PROGRAM Robot
VAR
	fbRobot						: FB_Robot_Mitsubishi;
	nCurrentState				: DINT;
	nLastState					: DINT;				
	rtRobot_ProgramStarted		: TON;
	rtRobot_ProgramCompleted	: TON;
	fbTimerRobot				:TON;
	gbTimerTimeoutRobot			:TON;
END_VAR

	Stations.gstRobotMitsubishi.sRobotAddress := '192.168.0.20';
	//gstRobotMitsubishi.bAutomaticMode := NOT IO_CONVEYOR.iMAINTENANCE_KEY;
	fbRobot(Robot := Stations.gstRobotMitsubishi,
		PacketManager := Stations.gstRobotMitsubishiPacketManager);
		
rtRobot_ProgramStarted(IN:=NOT Stations.gstRobotMitsubishi.bReady 
						AND NOT Stations.gstRobotMitsubishi.bProgramCompleted, PT:=T#50MS);
rtRobot_ProgramCompleted(IN:= Stations.gstRobotMitsubishi.bReady AND Stations.gstRobotMitsubishi.bProgramCompleted 
							AND Stations.gstRobotMitsubishi.nDependencyState = 0, PT:=T#10MS);

// If robot error
IF Stations.gstRobotMitsubishi.bError AND nCurrentState > E_RobotStates.STATE_INIT_CHECK_ROBOT_ERROR_DONE 
AND nCurrentState < E_RobotStates.STATE_ERROR THEN
	nLastState:=nCurrentState;
	nCurrentState:=E_RobotStates.STATE_ERROR;
END_IF
		
CASE nCurrentState OF
	E_RobotStates.STATE_WAITING_FOR_INIT:
		IF Stations.roboData = dataRequestRobot.roboInit THEN			
			nLastState := nCurrentState;
			nCurrentState := E_RobotStates.STATE_INIT_ROBOT_TOGGLE;
		END_IF
		
	E_RobotStates.STATE_INIT_ROBOT_TOGGLE:
		IF Stations.gstRobotMitsubishi.bAutomaticMode THEN
			Stations.gstRobotMitsubishi.bDoReset:=FALSE;
			Stations.gstRobotMitsubishi.bToggleConnect:=FALSE;
			Stations.gstRobotMitsubishi.bDoStart:=FALSE;
			fbTimerRobot(IN:=TRUE,PT:=T#1000MS);
			IF fbTimerRobot.Q THEN
				fbTimerRobot(IN:=FALSE);				
				nLastState := nCurrentState;
				nCurrentState :=E_RobotStates.STATE_INIT_ROBOT_ON;
			END_IF
		ELSE
			// Robot Auto  = true
		END_IF

	E_RobotStates.STATE_INIT_ROBOT_ON:
		IF Stations.gstRobotMitsubishi.bOnline THEN
			nLastState := nCurrentState;
			nCurrentState :=E_RobotStates.STATE_INIT_CHECK_ROBOT_ERROR;
		ELSE
			Stations.gstRobotMitsubishi.bToggleConnect:=TRUE;
			a_ToggleRobot();
		END_IF	

	E_RobotStates.STATE_INIT_CHECK_ROBOT_ERROR:
		IF Stations.gstRobotMitsubishi.bError OR Stations.gstRobotMitsubishi.nCurrentState = E_Robot_Mitsubishi_States.STATE_WAITING_RESET THEN
			Stations.gstRobotMitsubishi.bDoReset:=TRUE;
			nLastState := nCurrentState;
			nCurrentState :=E_RobotStates.STATE_INIT_CHECK_ROBOT_ERROR_DONE;
		ELSE
			nLastState := nCurrentState;
			nCurrentState :=E_RobotStates.STATE_INIT_CHECK_ROBOT_READY;
		END_IF	
	
	E_RobotStates.STATE_INIT_CHECK_ROBOT_ERROR_DONE:
		IF Stations.gstRobotMitsubishi.nCurrentState = E_Robot_Mitsubishi_States.STATE_OPERATIONAL THEN
			IF NOT Stations.gstRobotMitsubishi.bError THEN
				nLastState := nCurrentState;
				nCurrentState :=E_RobotStates.STATE_INIT_CHECK_ROBOT_READY;
			ELSE
				a_ToggleRobot();
			END_IF
		ELSIF Stations.gstRobotMitsubishi.nCurrentState = E_Robot_Mitsubishi_States.STATE_WAITING_RESET THEN
			nLastState := nCurrentState;
			nCurrentState :=E_RobotStates.STATE_INIT_CHECK_ROBOT_ERROR;
		END_IF
		
	E_RobotStates.STATE_INIT_CHECK_ROBOT_READY:
		IF NOT Stations.gstRobotMitsubishi.bReady OR NOT Stations.gstRobotMitsubishi.bExecuting THEN
			Stations.gstRobotMitsubishi.bDoStart:=TRUE;
			nLastState := nCurrentState;
			nCurrentState :=E_RobotStates.STATE_INIT_CHECK_ROBOT_READY_DONE;	
		ELSIF Stations.gstRobotMitsubishi.bBusy THEN
			Stations.gstRobotMitsubishi.bDoReset := TRUE;
			nLastState := nCurrentState;
			nCurrentState :=E_RobotStates.STATE_INIT_CHECK_ROBOT_BUSY;	
		ELSE
			nLastState := nCurrentState;
			nCurrentState :=E_RobotStates.STATE_INIT_CHECK_ROBOT_SERVOON;	
		END_IF
	
	E_RobotStates.STATE_INIT_CHECK_ROBOT_BUSY:
		gbTimerTimeoutRobot(IN:=TRUE,PT:=T#2000MS);
		IF Stations.gstRobotMitsubishi.nCurrentState = E_Robot_Mitsubishi_States.STATE_OPERATIONAL THEN
			gbTimerTimeoutRobot(IN:=FALSE);
			Stations.gstRobotMitsubishi.bDoStart := TRUE;
			nLastState := nCurrentState;
			nCurrentState :=E_RobotStates.STATE_INIT_CHECK_ROBOT_READY_DONE;
		ELSIF gbTimerTimeoutRobot.Q THEN
			gbTimerTimeoutRobot(IN:=FALSE);
			nLastState := nCurrentState;
			nCurrentState :=E_RobotStates.STATE_INIT_ROBOT_TOGGLE;
		END_IF
	
	E_RobotStates.STATE_INIT_CHECK_ROBOT_READY_DONE:
		IF Stations.gstRobotMitsubishi.bReady AND Stations.gstRobotMitsubishi.bExecuting THEN
			nLastState := nCurrentState;
			nCurrentState :=E_RobotStates.STATE_INIT_CHECK_ROBOT_SERVOON;
		ELSE
			a_ToggleRobot();					
		END_IF
				
	E_RobotStates.STATE_INIT_CHECK_ROBOT_SERVOON:		
		IF Stations.gstRobotMitsubishi.bPoweredOn AND Stations.gstRobotMitsubishi.bReady THEN
			nLastState := nCurrentState;
			nCurrentState :=E_RobotStates.STATE_INIT_DONE;
		ELSE 				
			Stations.gstRobotMitsubishi.bDoServoOn:=TRUE;
			nLastState := nCurrentState;
			nCurrentState :=E_RobotStates.STATE_INIT_CHECK_ROBOT_SERVOON_DONE;
		END_IF
		
	E_RobotStates.STATE_INIT_CHECK_ROBOT_SERVOON_DONE:
		IF Stations.gstRobotMitsubishi.bPoweredOn AND Stations.gstRobotMitsubishi.bReady THEN
			nLastState := nCurrentState;
			nCurrentState :=E_RobotStates.STATE_INIT_DONE;
		END_IF	
		
	E_RobotStates.STATE_INIT_DONE:
		Stations.roboData := dataRequestRobot.done;
		nLastState := nCurrentState;
		nCurrentState := E_RobotStates.STATE_WAITING_FOR_COMMAND;	
	
	E_RobotStates.STATE_WAITING_FOR_COMMAND:		
		IF Stations.roboData <> dataRequestRobot.done
		AND Stations.roboData <> dataRequestRobot.error THEN
			Stations.gstRobotMitsubishi.nTargetProgram := Stations.roboData;
			Stations.gstRobotMitsubishi.bDoStartProgram := TRUE;
			IF rtRobot_ProgramStarted.Q THEN
				nLastState := nCurrentState;
				nCurrentState := E_RobotStates.STATE_PROGRAM_DONE;
			END_IF
		END_IF
		
	E_RobotStates.STATE_PROGRAM_DONE:
		IF rtRobot_ProgramCompleted.Q THEN
			Stations.roboData := dataRequestRobot.done;
			nLastState := nCurrentState;
			nCurrentState := E_RobotStates.STATE_WAITING_FOR_COMMAND;
		END_IF
		
	E_RobotStates.STATE_ERROR:
		Stations.roboData := dataRequestRobot.error;
		nLastState := nCurrentState;
		nCurrentState := E_RobotStates.STATE_WAITING_FOR_INIT;
		
END_CASE

ACTION a_ToggleRobot:
fbTimerRobot(IN:=TRUE,PT:=T#2000MS);
IF fbTimerRobot.Q THEN
	fbTimerRobot(IN:=FALSE);
	nLastState := nCurrentState;
	nCurrentState :=E_RobotStates.STATE_INIT_ROBOT_TOGGLE;
END_IF
END_ACTION

END_PROGRAM

(* stored: Version 1.1.0.1, ProductVersion 3.1.4024.2
   POU ROBOT: Id {604af032-2a87-4ce8-af05-065565ae1cd2}, SpecialFunc None
   Action a_ToggleRobot: Id {93bc061d-ce6d-45c2-b967-a43187994360} *)
